// TIA Portal V20 export
DATA_BLOCK "IdentData"   // DB221
TITLE = Schnittstelle Read/Write Daten / Interface read/write data
AUTHOR : SICAR
FAMILY : Ident
VERSION : 1.0
// Ident Daten / Ident data
// stored: MemoryReserve 100
   VAR
      rfReader { ExternalAccessible := 'False'; ExternalVisible := 'False'; ExternalWritable := 'False'} : Array[0.."NO_OF_RF_IDENT_DEVICES"] of "LSicar_typeIdentReadWriteDat";   // Reader
   END_VAR
BEGIN
END_DATA_BLOCK
